INTERFACE ITF_PMLBase

METHOD SetStateComplete : BOOL
VAR_INPUT
END_VAR
END_METHOD

END_INTERFACE

(* stored: Version 1.1.0.1, ProductVersion 3.1.4024.11
   Itf ITF_PMLBase: Id {276ee589-9834-4be8-ac7c-1392e09b20b6}
   Method SetStateComplete: Id {f7d2376e-92b7-4e51-acb2-af71fe8c1c7c} *)
